FUNCTION_BLOCK CU050DialogContent EXTENDS TcoCore.TcoInputDialogContentContainer
VAR_INPUT
END_VAR
VAR_OUTPUT
END_VAR
VAR
	{attribute addProperty Name "<#Recipe#>"}
	Recipe:STRING;
	{attribute addProperty Name "<#Qantity#>"}
	RequiredQuantity:INT;
	{attribute addProperty Name "<#Timeout#>"}
	Timeout:DATE_AND_TIME;
	{attribute addProperty Name "<#Exclude#>"}
	Exclude:BOOL;

END_VAR

END_FUNCTION_BLOCK

(* stored: Version 1.1.0.1
   POU CU050DialogContent: Id {4db1f4a0-602a-4dab-982f-099c1b772cf4}, SpecialFunc None *)
